INTERFACE ITF

END_INTERFACE

(* stored: Version 1.1.0.1, ProductVersion 3.1.4024.16
   Itf ITF: Id {8971d2a1-f74c-41dc-9df2-63980a4f7ec8} *)
